Yaskawa INFORM job: TEST_BW.JBI

/JOB
//NAME TEST_BW
//POS
///NPOS 6,6,6,0,0,0
///TOOL 0
///POSTYPE PULSE
///PULSE
C00000=1999,-113620,-91817,15,89172,1
C00001=1999,-113620,-91817,15,89172,1
C00002=-135545,-89595,-39606,26842,74837,33039
C00003=-70479,-74327,-33913,25536,57772,53993
C00004=-73162,-72917,-36272,27270,63677,54011
C00005=-51396,-95630,-44793,25744,51293,59850
BC00000=87190,687249,787358
BC00001=343424,844605,787358
BC00002=343424,794511,527796
BC00003=343424,794511,527796
BC00004=343424,794511,527796
BC00005=343424,794511,527796
EC00000=1,0
EC00001=1,0
EC00002=1,0
EC00003=1,0
EC00004=1,0
EC00005=1,0
//INST
///DATE 2024/05/28 14:07
///ATTR SC,RW
///GROUP1 RB1,BS1
///GROUP2 ST1
NOP
MOVJ C00000 BC00000 VJ=100.00  +MOVJ EC00000 VJ=100.00
MOVJ C00001 BC00001 VJ=100.00  +MOVJ EC00001 VJ=100.00
MACRO1 MJ#(0) ARGF9
MOVL C00002 BC00002 V=166.7  +MOVJ EC00002 VJ=100.00
ARCON
MOVL C00003 BC00003 V=8.3  +MOVJ EC00003 VJ=100.00
ARCOF
MOVL C00004 BC00004 V=166.7  +MOVJ EC00004 VJ=100.00
MOVL C00005 BC00005 V=166.7  +MOVJ EC00005 VJ=100.00
END
